// TIA Portal V20 export
DATA_BLOCK "DB_Pressures"   // DB440
// stored: InstanceOfName FB_Pressures, InstanceOfType FB
"FB_Pressures"
   // VAR
   //    sTimeOutAirDryer : TON_TIME;
   //    sTimerMachineInDelay : TON_TIME;
   //    sTimeMachineReadyDelay { S7_SetPoint := 'True'} : TON_TIME;
   //    sAirInletPressureCtrl { S7_SetPoint := 'True'} : "FB_AnalogInputThreshold";
   //    sOverpressureScaleZ_Ctrl { S7_SetPoint := 'True'} : "FB_AnalogInputThreshold";
   //    sOverpressureOpticalPathCtrl { S7_SetPoint := 'True'} : "FB_AnalogInputThreshold";
   //    sOverpressureLaserHeadCtrl { S7_SetPoint := 'True'} : "FB_AnalogInputThreshold";
   //    sOverpressureAxisX_Y_Ctrl { S7_SetPoint := 'True'} : "FB_AnalogInputThreshold";
   // END_VAR
BEGIN
END_DATA_BLOCK
